TEXTLIST TextList_SA_Operations
  0 = 'Pompage' | FR: 'Pompage' | EN: 'Pumping'
  1 = 'Marche pompe' | FR: 'Marche\nPompes' | EN: 'Start\nPumps'
  2 = 'Arret pompe' | FR: 'Arrêt\nPompes' | EN: 'Stop\nPumps'
  3 = 'Isol' | FR: 'Isolement' | EN: 'Standby'
  4 = 'Vent' | FR: 'Ventilation' | EN: 'Venting'
  5 = 'Marche' | FR: 'Marche' | EN: 'Start'
  6 = 'Validation' | FR: 'Validation' | EN: 'Validation'
  7 = 'Arrêt' | FR: 'Arrêt' | EN: 'Stop'
  8 = 'Position' | FR: 'Positionnement' | EN: 'Positioning'
  9 = 'Initialisation' | FR: 'Repli' | EN: 'Folding'
  10 = 'cooling' | FR: "Refroidissement\nd'urgence" | EN: 'Emergency\nCooling'
  11 = 'pomp proc' | FR: 'Pompage\nProcédé' | EN: 'Process\nPumping'
  12 = 'on gaz' | FR: 'Mise en\ngaz' | EN: 'Start\ngas'
  13 = 'off gaz' | FR: 'Arrêt\ngaz' | EN: 'Stop\ngas'
  14 = 'rampee' | FR: 'Rampe\ngaz' | EN: 'Gas\nramp'
  15 = 'rotation' | FR: 'Rotation' | EN: 'Rotation'
  16 = 'Bal' | FR: 'Balayage' | EN: 'Sweeping'
  17 = 'regen' | FR: 'Régénération\nCryo' | EN: 'Cryo\nRegeneration'
  18 = 'charg' | FR: 'Chargement\nChambre' | EN: 'Chamber\nLoading'
  19 = 'decharg' | FR: 'Déchargement\nChambre' | EN: 'Chamber\nUnloading'
  20 = 'Init' | FR: 'Initialisation' | EN: 'Initialization'
  21 = 'Scan quartz' | FR: 'Scan quartz' | EN: 'Scan crystal'
  22 = 'Positionnement quartz' | FR: 'Positionnement quartz' | EN: 'Position crystal'
  23 = 'Position' | FR: 'Position' | EN: 'Position'
  24 = 'marche ch' | FR: 'Marche\nchauffage' | EN: 'Start\nheating'
  25 = 'arret ch' | FR: 'Arrêt\nchauffage' | EN: 'Stop\nheating'
  26 = 'Marche decap' | FR: 'Marche décapage' | EN: 'Start ion etching'
  27 = 'Stop decap' | FR: 'Arrêt décapage' | EN: 'Stop ion etching'
  28 = 'Pompage prim' | FR: 'Pompage\nprimaire' | EN: 'Primary\npumping'
  29 = 'Marche' | FR: 'Marche' | EN: 'Start'
   = ''
END_TEXTLIST

(* stored: Version 1.1.0.1, ProductVersion 3.1.4024.10
   TextList TextList_SA_Operations: Id {366ca346-e9df-42b4-bb8e-cf233c024502} *)
